(* PLC project Beremiz non-standard POUs library, Beremiz Beremiz 0.0 *)
(* stored: creationDateTime 2008-12-14T16:53:26, modificationDateTime 2019-08-06T14:08:26 *)

TYPE HMI_INT : INT;
END_TYPE

TYPE HMI_REAL : REAL;
END_TYPE

TYPE HMI_STRING : STRING;
END_TYPE

TYPE HMI_BOOL : BOOL;
END_TYPE

TYPE HMI_NODE : BOOL;
END_TYPE
